FUNCTION_BLOCK AND_BOOL (* IEC 61131-3 Boolean AND *)
  (* Standard: 61131-3 *)
  (* Version 0.0, 2004-12-15, JHC, Rockwell Automation, Converted from SRC format. *)
  (* Compiler header: package fb.rt.plc.bits; *)
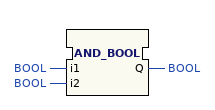
  VAR_INPUT
    i1 : BOOL;
    i2 : BOOL;
  END_VAR
  VAR_OUTPUT
    Q : BOOL;
  END_VAR
END_FUNCTION_BLOCK
